Staubli VAL3: onF8Event.pgx

program onF8Event(string x_sName (dimensions=1))
  local num l_nMax
begin
  // look if the bButton is enable
  if bButton[7]
    // NEXT
    call pallet:next(x_sName)
    // refresh it
    call buildList()
    use:bUseRefresh=true
  endIf
end
